// TwinCAT 3 PLC project plc
// ProgramVersion: 3.1.4024.0
// libraries:
//   Tc2_Standard, * (Beckhoff Automation GmbH)
//   Tc2_System, * (Beckhoff Automation GmbH)
//   Tc3_Module, * (Beckhoff Automation GmbH)
// project tree:
//   / GlobalTextList.TcGTLO, PlcTask.TcTTO, Visualization Manager.TcVMO (not stored)
//   GVLs/ Conc.TcGVL, Const.TcGVL, Flow.TcGVL, Status.TcGVL, Steam.TcGVL, Tank.TcGVL, Temp.TcGVL, UserIn.TcGVL, High.TcGVL
//   POUs/ RunAlarmCheck.TcPOU, RunFlash.TcPOU, RunSteam.TcPOU, RunTime.TcPOU, SetCIP.TcPOU, NextConc.TcPOU, MAIN.TcPOU, NextHigh.TcPOU, GetReactRate.TcPOU, NextTemp.TcPOU, GetVolume.TcPOU, GetOutFlow.TcPOU
//   VISUs/ Vis.TcVIS, WIP.TcVIS
// real-time tasks:
//   TASK PlcTask: cycle T#10ms, priority 20, ADS port 350

CONFIGURATION plc
    RESOURCE PLC ON TwinCAT3
        TASK PlcTask(INTERVAL := T#10ms, PRIORITY := 20);
        PROGRAM MAIN WITH PlcTask : MAIN;
    END_RESOURCE
END_CONFIGURATION

// ---- GVLs/Conc.TcGVL
{attribute 'qualified_only'}

// CONCENTRATION [mol/m3]

VAR_GLOBAL
	
	// Current concentration 
	now : REAL := 1.0;
	
	// Concentration in
	in  : REAL := 10;
	
END_VAR

VAR_GLOBAL CONSTANT
	
	// CIP, Normal concentration in
	cip    : REAL :=  5;
	normal : REAL := 10;
	
END_VAR

// ---- GVLs/Const.TcGVL
{attribute 'qualified_only'}

// CONSTANT VALUES

VAR_GLOBAL CONSTANT
	
	// Gravitational acceleration [N/kg]
	grav : REAL := 9.81;
	
	// Activation Energy [K]
	AE   : REAL := 5000;

	// Rate Konstant [m3/mol/s] (as opposed to the Rate *C*onstant?)		
	Rk   : REAL := 578000;

	// Density of the liquid [kg/m3]
	rho  : REAL := 1000;
	
	// Thermal transfer Koefficient [J/s/K/m2] (again with the *K*?)
	Kwall : REAL := 600;

	// Specific heat of the liquid [J/kg/K]
	cp   : REAL := 4180;

	// Heat of Reaction [J/mol]
	Hr   : REAL := 45000;

END_VAR

// ---- GVLs/Flow.TcGVL
{attribute 'qualified_only'}

// FLOW [m3/s]

VAR_GLOBAL
	
	// Inlet flow
	in  : REAL := 0.002; // This one seems to set itself to 0...
	
	// Outlet flow (indicative only - is calculated externally)
	out : REAL := 0;
	
END_VAR

VAR_GLOBAL CONSTANT
	
	// CIP & normal flows
	cip    : REAL := 0.004;
	normal : REAL := 0.002;
	
END_VAR

// ---- GVLs/Status.TcGVL
{attribute 'qualified_only'}

// STATUS & SIMULATION VARS

VAR_GLOBAL
	
	// CIP status
	is_cip : BOOL := FALSE;
	
	// Alarm status
	alarm : BOOL := FALSE;
		
	// Time now and time per machine cycle
	time_now  : REAL := 0; // [s]
	
	// Flash generator
	flash : BOOL := FALSE;
	
END_VAR

VAR_GLOBAL CONSTANT
	
	// CIP period
	time_cip : REAL := 20 *60; // [s]
	
	// CIP cycle period
	time_cycle : REAL := 2 *60 *60; // [s]
		
END_VAR

// ---- GVLs/Steam.TcGVL
{attribute 'qualified_only'}

// STEAM [°C]

VAR_GLOBAL
	
	// Current steam tempurature
	now    : REAL := 50;
	
	// Target steam tempurature
	target : REAL := 50;
		
END_VAR

VAR_GLOBAL CONSTANT
	
	// Minimum, Maximum, Tempurature change per second
	mini : REAL :=  50;
	maxi : REAL := 300;
	step : REAL :=  10; // change per second
	
END_VAR

// ---- GVLs/Tank.TcGVL
{attribute 'qualified_only'}

// TANK PROPERTIES [m, m2, m3]

VAR_GLOBAL CONSTANT
	
	D : REAL := 1.8;
	H : REAL := 2.5;
	A : REAL := PI * EXPT(D, 2) / 4;
	V : REAL := A * H;
	
END_VAR

// ---- GVLs/Temp.TcGVL
{attribute 'qualified_only'}

// TEMPURATURE [°C]

VAR_GLOBAL
	
	// Current tempurature
	now  : REAL := 80;
	
	// Wall temp
	wall : REAL := 25;
	
END_VAR

VAR_GLOBAL CONSTANT
	
	// Inlet temp (const)
	in : REAL := 25;
	
	// Offset for Celcius/Kelvin conversion
	offset : REAL := 273.16;
	
END_VAR

// ---- GVLs/UserIn.TcGVL
{attribute 'qualified_only'}

// USER INPUTS

VAR_GLOBAL
	
	// Time step [s]
	time_step    : REAL := 2;
	
	// Outlet valve position [0-100 as percentage]
	out_percent  : REAL := 0;
	
	// Steam tempurature [°C]
	steam_temp   : REAL := 50;
	
	// Autohold status
	IO_match     : BOOL := FALSE;
	
	// Stop buttons
	enable_in    : BOOL := TRUE;
	enable_steam : BOOL := TRUE;
	
END_VAR

// ---- GVLs/High.TcGVL
{attribute 'qualified_only'}

// HEIGHT [m]

VAR_GLOBAL
	
	// Current height
	now : REAL := 2.2;
	
	// Current level in tank as percentage
	full_percent : REAL := 0; // [0-100.1%] (small overflow)
	
END_VAR

// ---- POUs/MAIN.TcPOU
PROGRAM MAIN

VAR
	h : REAL;
	t : REAL;
	c : REAL;
END_VAR

// Run all calculations on same data - save new values at end of machine cycle
h := NextHigh();
t := NextTemp();
c := NextConc();

// Update the globals
High.now := h;
Temp.now := t;
Conc.now := c;

// Run steam
RunSteam();

// Run alarm
RunAlarmCheck();

// Run time
RunTime();

// Run flash
RunFlash();

END_PROGRAM

// ---- POUs/NextHigh.TcPOU

// CALCULATE THE NEXT HEIGHT OF LIQUID IN THE TANK

FUNCTION NextHigh : REAL

VAR
	
	// Flow in [m3/s]
	in : REAL := flow.in;
	
	// Flow out [m3/s]
	out : REAL := GetOutFlow();
	
	// Coeff [s/m2]
	coef : REAL := userin.time_step / tank.A;
	// s / m2 -> s/m2
	
	// delta [m]
	dhigh : REAL;
	// m3/s * s/m2 -> m
	
	// Truncate the maximum height
	maxi : REAL := tank.H * 1.001;
	
	// Temporary variable to hold the next value
	next : REAL;

END_VAR

// Calculate the next height
dhigh := (in - out) * coef;
next := High.now + dhigh;

// Remove overflow and error handling
IF next > maxi THEN
	next := maxi;
ELSIF next <= 0 THEN
	next := 0;
END_IF

// Return next height
NextHigh := next;

// Update the fullnes percentage
High.full_percent := next * 100 / tank.H;

END_FUNCTION

// ---- POUs/GetOutFlow.TcPOU

// CALCULATE THE CURRENT OUTFLOW [m3/s]

FUNCTION GetOutFlow : REAL

VAR
	// Module A []
	a : REAL := 14 * EXPT(10,-6);
	
	// Module B []
	b : REAL := SQRT(2 * const.grav * High.now);
	
	// Combine MA and MB []
	coef : REAL := a * b;
	
	
	// Outlet valve value [0-100%]
	valve : REAL := userin.out_percent;

	// Flow in and out [m3/s]
	in  : REAL := flow.in;
	out : REAL;
	
	// Auto hold is enabled?
	match : BOOL := userin.IO_match;

END_VAR

// Calculate output
out := coef * valve;

IF out < 0 THEN
	out := 0;
END_IF

// Return flow value
GetOutFlow := out;
flow.out := out;

// If running IO matching
// Try to find a valve setting to equate in and out
IF match THEN
	userin.out_percent := valve + (in-out)*1000;
END_IF

END_FUNCTION

// ---- POUs/NextTemp.TcPOU

// CALCULATE THE NEXT TEMPURATURE OF THE LIQUID

FUNCTION NextTemp : REAL

VAR
	
	// // Heat in [J/s] // //
	a : REAL := const.rho * flow.in * const.cp;
	// kg/m3 * m3/s * J/kg/K -> J/s/K
	
	b : REAL := temp.in - temp.now;
	// K - K -> K
	
	Qin : REAL := a * b;
	// J/s/K * K -> J/s
	
	
	// // Heat from reaction [J/s]	// //
	
	Qre : REAL := GetReactRate() * GetVolume() * const.Hr;
	// mol/m3/s * m3 * J/mol -> J/s
	
	
	// // Heat conducted in from steam jacket [J/s] // //
	
	c   : REAL := const.Kwall * tank.D * PI * High.now;
	// J/s/K/m2 * m * m -> J/s/K
	
	d   : REAL := temp.wall  - temp.now;
	// K - K -> K
	
	Qco : REAL := c * d;
	// J/s/K * K -> J/s
	
	
	// // Support coefficients // //

	dtime : REAL := userin.time_step;
	// s
	
	mtcp  : REAL := const.rho * const.cp * GetVolume();
	// kg/m3 * J/kg/K * m3 -> J/K
	
	
	// // Delta [K] // //
	dtemp : REAL;
	// J/s * s / J/K -> K
	
END_VAR

// Throw error
IF mtcp <= 0 THEN
	nexttemp := 0;
	RETURN;
END_IF

dtemp := (Qin + Qre + Qco) * dtime / mtcp;
NextTemp := temp.now + dtemp;

END_FUNCTION

// ---- POUs/GetReactRate.TcPOU

// CALCULATE CURRENT REACTION RATE [mol/m3/s]

FUNCTION GetReactRate : REAL

VAR
	
	// Module A [(mol/m3)2]
	a : REAL := EXPT(Conc.now,2); 
	
	// Module B [m3/mol/s]
	b : REAL := Const.Rk; 
	
	// Module C []
	kelvin : REAL := temp.now + temp.offset;
	AE     : REAL := const.AE;
	c      : REAL;
	
END_VAR

// Error handling
IF kelvin <= 0 THEN
	getreactrate :=0;
	RETURN;
END_IF

c := EXP(-AE / kelvin);

// [mol2/m32 * m3/mol/s -> mol/m3/s]
GetReactRate := a * b * c;

END_FUNCTION

// ---- POUs/GetVolume.TcPOU

// GET THE CURRENT VOLUME OF LIQUID IN THE TANK [m3]

FUNCTION GetVolume : REAL

VAR
	
	a : REAL := tank.A;
	h : REAL := High.now;
	
END_VAR

GetVolume := a * h;

END_FUNCTION

// ---- POUs/NextConc.TcPOU

// CALCULATE THE NEXT CONCENTRATION VALUE [mol/m3]

FUNCTION NextConc : REAL

VAR
	
	// Concentration in [mol/s]
	in : REAL := conc.in * flow.in;
	// mol/m3 * m3/s -> mol/s
	
	// Conc destroyed [mol/s]
	des : REAL :=  GetReactRate() * GetVolume();
	// mol/m3/s * m3 -> mol/s
	
	// Conc out [mol/s]
	out : REAL := conc.now * getoutflow();
	// mol/m3 * m3/s -> mol/s
	
	// Coefficient
	step : REAL := userin.time_step;
	vol  : REAL := GetVolume();
	// step/vol -> s/m3
	
	// delta  [mol/m3]
	dconc : REAL;
	// mol/s * s/m3 -> mol/m3
	
END_VAR

// Throw error
IF vol = 0 THEN
	NextConc := 0;
	RETURN;	
END_IF

dconc := (in - des - out) * step / vol;

IF dconc > 0 THEN
	dconc := 0;
END_IF

NextConc := conc.now + dconc;

END_FUNCTION

// ---- POUs/RunSteam.TcPOU

// CALCULATE NEXT STEAM TEMPURATURE

FUNCTION RunSteam

VAR
	
	// User input target
	targ : REAL := userin.steam_temp;
	enabled : bool := userin.enable_steam;
	
	// Import steam parameters for clarity
	now  : REAL := steam.now;
	maxi : REAL := steam.maxi;
	mini : REAL := steam.mini;
	step : REAL := steam.step * userin.time_step;
	
	// Calculation variables
	new  : REAL;
	diff : REAL;
	
END_VAR

// Import target temp from GUI
steam.target := targ;

// Validation
IF step <= 0 THEN
	RETURN;
ELSIF targ > maxi THEN
	targ := maxi;
ELSIF targ < mini THEN
	targ := mini;
END_IF

// Manual override
IF NOT enabled THEN
	targ := 20;
END_IF


// Calculate what change is needed to meet the target
diff := targ - now;


// LESS than target and MORE than a step away
IF diff >= step THEN
	// New temp is this plus step
	new := now + step;	

// GREATER then target and MORE than a step away
ELSIF diff <= -step THEN
	// New temp is this minus step
	new := now - step;

// Is correct or within one step
ELSE
	new := targ;
END_IF

// Save new value
temp.wall := new;
steam.now := new;

END_FUNCTION

// ---- POUs/RunAlarmCheck.TcPOU

// RUN THE ALARM CHECK

FUNCTION RunAlarmCheck

VAR
	// Threashold value (both tests just happen to use the same value)
	thresh : REAL := 90;
	
	// FILL is alarm?
	h : BOOL := High.full_percent > thresh;
	
	// TEMP is alarm?
	t : BOOL := Temp.now > thresh;
	
END_VAR

status.alarm := h OR t;

END_FUNCTION

// ---- POUs/RunTime.TcPOU

// PROCESS THIS MACHINE CYCLE AS A TIME STEP

FUNCTION RunTime

VAR
	
	// Read in values for easy access
	cycle : REAL := status.time_cycle;
	step  : REAL := userin.time_step; 
	next  : REAL := status.time_now + step;
	cip   : REAL := cycle - status.time_cip;	
	
END_VAR

IF step <= 0 THEN
	RETURN;
END_IF

// Loop back to 0 if new time is over
IF next > cycle THEN
	next := 0;
END_IF

// Update CIP status based on the new time
SetCIP(next >= cip);

// Save new time
status.time_now := next;

END_FUNCTION

// ---- POUs/SetCIP.TcPOU

// SET THE CLEAN-IN-PLACE STATUS

FUNCTION SetCIP

VAR_INPUT
	
	// New CIP status
	cip : BOOL := FALSE;
	
END_VAR

VAR
	
	// Inlet enabled status
	enable : BOOL := userin.enable_in;
	
END_VAR

// I'd love a ternary operator about now...

// If in manual override
IF NOT enable THEN
	flow.in := 0;
	status.is_cip := FALSE;
	RETURN;
	
// If currently CIP -> set appropriate values	
ELSIF cip THEN
	conc.in := conc.cip;
	flow.in := flow.cip;
	
// Otherwise, set the normal values
ELSE
	conc.in := conc.normal;
	flow.in := flow.normal;
END_IF

// Update status value
status.is_cip := cip;

END_FUNCTION

// ---- POUs/RunFlash.TcPOU

// RUN THE FLASH CALC

FUNCTION RunFlash

VAR
	
	time_now  : INT := REAL_TO_INT(status.time_now);
	time_step : INT := REAL_TO_INT(userin.time_step);
	
	// Current machine cycle
	macy_now  : INT;
	flcy_now  : INT;
	
	// Number of machine cycles per flash cycle
	macy_per_flcy : INT := 10;
	duty_cycle_pc : INT := 90;

END_VAR

IF time_step <= 0 THEN
	RETURN;
END_IF

macy_now := time_now / time_step;

flcy_now := macy_now MOD macy_per_flcy;

status.flash := flcy_now < macy_per_flcy *duty_cycle_pc/100;

END_FUNCTION

// ---- GlobalTextList.TcGTLO
TEXTLIST GlobalTextList
  134 = ''
  264 = '                                             THING'
  277 = '                    THING'
  863 = '                 C.I.P. RUNNING'
  47 = '                 INLET ENABLE'
  942 = '                 MASTER ALARM'
  183 = '                 STEAM ENABLE'
  141 = '                C.I.P. RUNNING'
  854 = '            C.I.P. RUNNING'
  875 = '            Clean In Place'
  625 = '          THING'
  851 = '%'
  546 = '%.1*100f'
  168 = '%.1f'
  501 = '%.1f*100'
  9 = '%.1fmol/m³'
  918 = '%.1i'
  57 = '%.1r'
  606 = '%.2f'
  631 = '%1*f'
  506 = '%1.0f'
  48 = '%1.1f'
  964 = '%1f'
  819 = '%2.1i'
  466 = '%2d'
  601 = '%2d%%'
  137 = '%d00 L'
  583 = '%f'
  285 = '%GVL.time_now'
  570 = '%i'
  922 = '%i%%'
  608 = '%i*100'
  656 = '%i°C'
  166 = '%s'
  411 = 'adf \nadf'
  21 = 'adf $n adf'
  778 = 'adf \\n adf'
  596 = 'adf$nadf'
  417 = 'CLEAN IN PLACE'
  418 = 'conc mol/m³'
  83 = 'Conc.: %1.2f mol/m3'
  661 = 'Conc: %1.2f mol/m3'
  681 = 'Conc: %2.2f mol/L'
  706 = 'Conc: %2.2f mol/m3'
  728 = 'conc\\nmol/m³'
  1 = 'Flow: %1.2f'
  272 = 'Flow: %1.2f L/s'
  634 = 'Flow: %2.2f L/s'
  782 = 'Flow: %f.2'
  584 = 'Flow: %f0.2'
  290 = 'Flow: %f1.2'
  883 = 'GVL.time_now'
  284 = 'i'
  169 = 'I/O HOLD'
  638 = 'I/O MATCH'
  390 = 'INFORMATION'
  679 = 'INLET'
  760 = 'INLET %i %i'
  816 = 'INLET ENABLE'
  999 = 'INLET/N'
  595 = 'MASTER ALERT'
  182 = 'mol/L'
  399 = 'mol/m³'
  93 = 'Now: %d s'
  126 = 'OUTLET'
  831 = 'OVER\nFLOW'
  626 = 'OVER\nHEAT'
  741 = 'OVER $L FLOW'
  900 = 'OVER$L FLOW'
  624 = 'OVER$LFLOW'
  412 = 'OVER$nFLOW'
  473 = 'OVER$NFLOW'
  111 = "OVER'$nFLOW"
  96 = 'OVERFLOW'
  657 = 'OVERHEAT'
  334 = 'STEAM'
  386 = 'Step: %d s'
  374 = 'Temp: %1.2f L/s'
  472 = 'Temp: %2.2f °C'
  680 = 'THING'
  138 = 'TIME CONTROL'
  231 = 'Time: %i'
  571 = 'Volume: %d00 L'
  655 = 'Volume: %d000 L'
  794 = 'X10°C'
  230 = '°C'
  774 = '°C*10'
END_TEXTLIST

// ---- VISUs/Vis.TcVIS
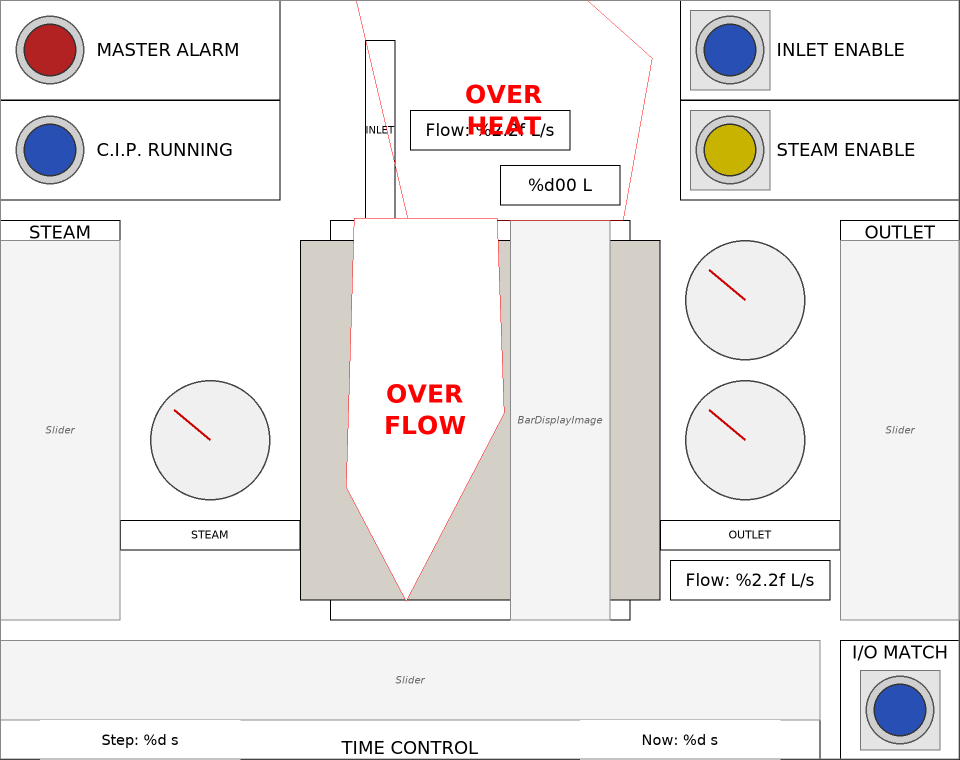
VISUALIZATION Vis  // 960x760
    Rectangle (0,0 960x760)
    Rectangle (670,560 160x40), "Flow: %2.2f L/s", text variable: Flow.out*1000
    Rectangle (660,520 180x30), "OUTLET"
    Rectangle (290,115 180x30), angle 90, "INLET"
    Rectangle (120,520 180x30), "STEAM"
    Group (840,220 120x400)
        Rectangle (0,0 120x400), "OUTLET"
        Slider (0,20 120x380), variable: UserIn.out_percent, scale 0..100
            p2985826283: %i%%
    Group (0,220 120x400)
        Rectangle (0,0 120x400), "STEAM"
        Slider (0,20 120x380), variable: UserIn.steam_temp, scale 0..100
            p2985826283: %i°C
    Meter360 (150,380 120x120), value: steam.now, style: Meter-Meter360-Yellow, scale format: %i, scale 0..350
        p518627256: °C
    Group (840,640 120x120)
        Rectangle (0,0 120x120), "I/O MATCH"
        PushSwitchLed (20,30 80x80), variable: UserIn.IO_match, behaviour: TOGGLE, style: Switch-PushSwitchLed-Blue
    Group (300,220 360x400)
        Rectangle (30,0 300x400)
        RoundedRectangle (0,20 360x360)
    BarDisplayImage (510,220 100x400), value: High.full_percent, style: BarDisplayImage-Gray, scale format: %2d%%, scale 0..100
    Meter360 (685,240 120x120), value: temp.now, style: Meter-Meter360-Blue, scale format: %i, scale 0..120
        p518627256: °C
    Meter360 (685,380 120x120), value: conc.now*100, style: Meter-Meter360-Green, scale format: %1.1f, scale 0..10
        p518627256: mol/m³
    Group (0,0 280x200)
        OnMouseClick: execute {
            userin.out_percent := 100;
            userin.steam_temp := steam.mini;
            userin.IO_match := FALSE;
        }
        Group (0,100 280x100)
            Rectangle (0,0 280x100), "C.I.P. RUNNING"
            Lamp1 (10,10 80x80), variable: Status.is_cip, style: Lamp-Lamp1-Blue
        Group (0,0 280x100)
            Rectangle (0,0 280x100), "MASTER ALARM"
            Lamp1 (10,10 80x80), variable: Status.alarm, style: Lamp-Lamp1-Red
    Group (0,640 820x120)
        Rectangle (0,0 820x120), "TIME CONTROL"
        Slider (0,0 820x80), variable: UserIn.time_step, scale 0..100
        Rectangle (40,80 200x40), "Step: %d s", text variable: UserIn.time_step
        Rectangle (580,80 200x40), "Now: %d s", text variable: Status.time_now
    Rectangle (410,110 160x40), "Flow: %2.2f L/s", text variable: Flow.in*1000
    Rectangle (500,165 120x40), "%d00 L", text variable: Tank.A * High.now * 10
    Polygon (408,220) (356,0) (587,0) (652,58) (623,220), "OVER HEAT", invisible if: Temp.now <= 100
        OnMouseClick: execute {
            userin.out_percent := 100;
            userin.steam_temp := steam.mini;
            userin.IO_match := FALSE;
        }
    Polygon (354,218) (497,218) (504,413) (406,601) (346,487), "OVER FLOW", invisible if: High.full_percent <=100
        OnMouseClick: execute { userin.out_percent := 100; userin.IO_match := FALSE; }
    Group (680,0 280x200)
        Group (0,100 280x100)
            Rectangle (0,0 280x100), "STEAM ENABLE"
            PushSwitch (10,10 80x80), variable: UserIn.enable_steam, behaviour: TOGGLE, style: Switch-PushSwitch-Yellow
        Group (0,0 280x100)
            Rectangle (0,0 280x100), "INLET ENABLE"
            PushSwitch (10,10 80x80), variable: UserIn.enable_in, behaviour: TOGGLE, style: Switch-PushSwitch-Blue
END_VISUALIZATION

// ---- VISUs/WIP.TcVIS
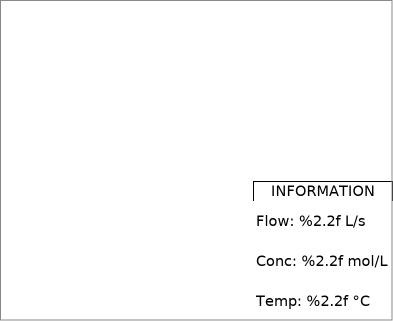
VISUALIZATION WIP  // 393x321
    Group (253,181 140x140)
        Rectangle (0,0 140x140), "INFORMATION"
        Rectangle (0,20 140x40), "Flow: %2.2f L/s", text variable: Flow.out*1000
        Rectangle (0,60 140x40), "Conc: %2.2f mol/L", text variable: Conc.now*1000
        Rectangle (0,100 140x40), "Temp: %2.2f °C", text variable: Temp.now
END_VISUALIZATION
